FUNCTION_BLOCK FB_OutOfService IMPLEMENTS I_State
VAR_INPUT
	(* Pointer to the ATM Machine*)
	pATM_Machine	: POINTER TO FB_ATM_Machine;
END_VAR
VAR_OUTPUT
END_VAR
VAR
END_VAR

METHOD Cancel : BOOL
END_METHOD

METHOD Card_Ejected : BOOL
END_METHOD

METHOD Card_Inserted : BOOL
END_METHOD

PROPERTY Description : E_StateDescription
GET
Description := E_StateDescription.OutOfService;
END_GET
END_PROPERTY

METHOD Failure : BOOL
END_METHOD

METHOD FB_Init : BOOL
VAR_INPUT
	(* if TRUE, the retain variables are initialized (warm start / cold start)*)
	bInitRetains	: BOOL;
	(* if TRUE, the instance afterwards gets moved into the copy code (online change)*)
	bInCopyCode	: BOOL;
	(* Pointer to the ATM Machine*)
	pATM_Machine	: POINTER TO FB_ATM_Machine;
END_VAR
THIS^.pATM_Machine := pATM_Machine;
END_METHOD

METHOD Op : BOOL
END_METHOD

METHOD Service : BOOL
ADSLOGSTR(ADSLOG_MSGTYPE_LOG, 'Entering Service Mode...', '');
pATM_Machine^.SetState(pATM_Machine^.MaintenanceState);
END_METHOD

METHOD SystemTest_OK : BOOL
END_METHOD

METHOD Turn_Off : BOOL
ADSLOGSTR(ADSLOG_MSGTYPE_LOG, 'Turning off machine...', '');
pATM_Machine^.SetState(pATM_Machine^.OffState);
END_METHOD

METHOD Turn_On : BOOL
END_METHOD

END_FUNCTION_BLOCK

(* stored: Version 1.1.0.1, ProductVersion 3.1.4024.12
   POU FB_OutOfService: Id {723d3d50-c51c-08c6-01e3-ca5a3f6f5f5f}, SpecialFunc None
   Method Cancel: Id {9ffe729a-ed4e-0074-2a78-fee68c1f05b2}
   Method Card_Ejected: Id {6c51b482-94c3-0ac6-388a-851186b19f5c}
   Method Card_Inserted: Id {56da786d-000b-02e7-17cf-16c9f8c4ec56}
   Property Description: Id {b4293c98-a8e6-0fdb-1621-a432f1054519}
   Get Get: Id {c4da1f8e-7da0-0f66-187d-a0b1bc68a431}
   Method Failure: Id {03454216-0922-0640-3f7d-0ed5f7654e0b}
   Method FB_Init: Id {fa6e6e68-dffe-0117-26d8-96e73a09489f}
   Method Op: Id {ea83443f-7c7a-0814-0a64-8bc75d8f7a89}
   Method Service: Id {f04780a3-6783-0dbc-266b-0f86bf43f3b3}
   Method SystemTest_OK: Id {da0693fd-4085-035f-3b0d-a3f82054f4ae}
   Method Turn_Off: Id {edd42c42-d61c-0274-0331-67a0e8de7e58}
   Method Turn_On: Id {83b4a46b-df13-0cc0-140b-518fc5d203ec} *)
